// TwinCAT 3 PLC project Untitled1
// ProgramVersion: 3.1.4024.0
// libraries:
//   Tc2_Standard, * (Beckhoff Automation GmbH)
//   Tc2_System, * (Beckhoff Automation GmbH)
//   Tc3_Module, * (Beckhoff Automation GmbH)
// project tree:
//   DUTs/ TYP_BUTTONS_HW_IN.TcDUT, TYP_VESSEL_HW.TcDUT, TYP_VESSEL_HW_IN.TcDUT, TYP_VESSEL_HW_OUT.TcDUT
//   GVLs/ gOpc.TcGVL
//   / PlcTask.TcTTO
//   POUs/ MAIN.TcPOU, VesselControlFB.TcPOU
// real-time tasks:
//   TASK PlcTask: cycle T#10ms, priority 20, ADS port 350

CONFIGURATION Untitled1
    RESOURCE PLC ON TwinCAT3
        TASK PlcTask(INTERVAL := T#10ms, PRIORITY := 20);
        PROGRAM MAIN WITH PlcTask : MAIN;
    END_RESOURCE
END_CONFIGURATION

// ---- DUTs/TYP_BUTTONS_HW_IN.TcDUT
TYPE TYP_BUTTONS_HW_IN :
STRUCT
	ModeButton : BOOL; // false - state = MANUAL; true - state = AUTOMATIC
	AnalogButtons : ARRAY [1..2] OF INT; // in manual mode button 1 = Max value for vessel 2 pressure; 2 = Min value for vessel 2 pressure
END_STRUCT
END_TYPE

// ---- DUTs/TYP_VESSEL_HW.TcDUT
TYPE TYP_VESSEL_HW :
STRUCT
	In : TYP_VESSEL_HW_IN;
	Out : TYP_VESSEL_HW_OUT;
END_STRUCT
END_TYPE

// ---- DUTs/TYP_VESSEL_HW_IN.TcDUT
TYPE TYP_VESSEL_HW_IN :
STRUCT
	Sensor : INT; //pressure of the vessel
END_STRUCT
END_TYPE

// ---- DUTs/TYP_VESSEL_HW_OUT.TcDUT
TYPE TYP_VESSEL_HW_OUT :
STRUCT
	Valves : BOOL; //vessel valve true = open; false = closed
END_STRUCT
END_TYPE

// ---- GVLs/gOpc.TcGVL
{attribute 'qualified_only'}
VAR_GLOBAL
	{attribute 'OPC.UA.DA' := '1'}
	Vessel : ARRAY [1..2] OF TYP_VESSEL_HW;
	{attribute 'OPC.UA.DA' := '1'}
	Buttons : TYP_BUTTONS_HW_IN;
	{attribute 'OPC.UA.DA' := '1'}
	SystemState : INT;	
END_VAR

// ---- POUs/MAIN.TcPOU
PROGRAM MAIN
VAR
VesselControll_Program :	VesselControlFB ;
END_VAR

VesselControll_Program();

END_PROGRAM

// ---- POUs/VesselControlFB.TcPOU
FUNCTION_BLOCK VesselControlFB
VAR_INPUT	
END_VAR
VAR_OUTPUT	
END_VAR
VAR			
iPressureLimitVessel_2_Min : INT; 		//Temp Variables for Vessel2 Pressure Control 
iPressureLimitVessel_2_Max : INT; 		//Temp Variables for Vessel2 Pressure Control 	
AutoManPushButton_rTrig : R_TRIG ;			//Button Rise Edge Read
END_VAR
VAR CONSTANT 
cAutoLimitMinPressureVessel2 : INT :=40; // Automatic Pressure Control Constant MIN
cAutoLimitMaxPressureVessel2 : INT :=60; // Automatic Pressure Control Constant MAX
cOneBar : INT :=1;						// Constant 1 Bar 
iAutoMode : INT := 1;
iManualMode : INT := 0;
END_VAR

//=============================================================================
// Dmitri Raihtsaum - Copyright 2023
// Created By: Dmitri Raihtsaum
//-----------------------------------------------------------------------------
// Tested with:   Twincat3, UaExpert
// Engineering:   Twincat3
// Functionality: Test Home Work - Vessel Pressure Control
// Date: 20.07.2023
// Rev 0.1
//=============================================================================

AutoManPushButton_rTrig(CLK :=  gOpc.Buttons.ModeButton); 		//Button Rise Edge Read
// System Mode Control
// push button for toggling the state between AUTOMATIC and MANUAL.
IF AutoManPushButton_rTrig.Q AND gopc.SystemState = iAutoMode THEN  			//Change From Auto To Manual
	gopc.SystemState := iManualMode;											//Change From Auto To Manual
ELSIF AutoManPushButton_rTrig.Q AND gopc.SystemState = iManualMode THEN		//Change From Manual To Auto
	gopc.SystemState:= iAutoMode; 											//Change From Manual To Auto
END_IF;
//Vessel 1 Control
// The pressure must be equal in both vessels ± 1 bar.
// Pressure in Vessel 1 is controlled in reference to Vessel 2 pressure:
// When pressure in Vessel 1 is 1 bar higher than is Vessel 2, then the Vessel 1
//valve shall be opened to release the pressure until the pressure in Vessel 1
//in 1 bar lower than the pressure in Vessel 2.

IF gOpc.Vessel[1].In.Sensor  >=  gOpc.Vessel[2].In.Sensor + cOneBar  THEN // Pressure Comparation Vessel1 and Vessel2 
	gOpc.Vessel[1].Out.Valves  :=TRUE;									  //Open Valve Y1
END_IF;

IF gOpc.Vessel[1].In.Sensor  <=  gOpc.Vessel[2].In.Sensor - cOneBar  THEN // Pressure Comparation Vessel1 and Vessel2
	gOpc.Vessel[1].Out.Valves  := FALSE;								  //Close Valve Y1
END_IF;
//Vessel 2 Control
//• Pressure in Vessel 2 is controlled in REFERENCE TO MIN AND MAX pressure
//parameters:
//o When pressure in Vessel 2 reaches Max parameter, then the Vessel 2 valve
//shall be opened to release the pressure until the pressure in Vessel 2
//reaches Min parameter.
//• The system shall have 2 states:
//o AUTOMATIC Min and Max parameters for Vessel 2 are given as
//constants 40 bar and 60 bar correspondingly.
//o MANUAL Min and Max parameters for Vessel 2 are given by Button 1
//(analogue potentiometer knob) and Button 2 (analogue potentiometer
//knob).
//o The state shall be changed using a third button (push button).
IF gopc.SystemState= iManualMode THEN 
	iPressureLimitVessel_2_Min := gOpc.Buttons.AnalogButtons[1];   //Temp Varibles data sellection
	iPressureLimitVessel_2_Max := gOpc.Buttons.AnalogButtons[2];	//Temp Varibles data sellection
END_IF;
IF gopc.SystemState = iAutoMode THEN 
	iPressureLimitVessel_2_Min := cAutoLimitMinPressureVessel2;			//Temp Varibles data sellection
	iPressureLimitVessel_2_Max := cAutoLimitMaxPressureVessel2;			//Temp Varibles data sellection
END_IF;
IF gOpc.Vessel[2].In.Sensor  >= iPressureLimitVessel_2_Max THEN  // Pressure Comparation  Vessel2 and Limits
	gOpc.Vessel[2].Out.Valves  :=TRUE;												//Open Valve Y2
END_IF
IF gOpc.Vessel[2].In.Sensor <= iPressureLimitVessel_2_MIN THEN // Pressure Comparation  Vessel2 and Limits
	gOpc.Vessel[2].Out.Valves  :=FALSE;											//Close Valve Y2
END_IF

//=============================================================================
//END
//=============================================================================

END_FUNCTION_BLOCK
